// TIA Portal V17 export
// export: Created 2023-04-11T09:33:31.0535455Z, ExportSetting WithDefaults, DisplayName Totally Integrated Automation Portal, DisplayVersion V17 Update 3, DisplayName TIA Portal Openness, DisplayVersion V17 Update 3, DisplayName TIA Portal Version Control Interface, DisplayVersion V17, DisplayName SINAMICS Startdrive Advanced, DisplayVersion V17 Update2, DisplayName SINAMICS Startdrive G130, G150, S120, S150, SINAMICS MV, S210, DisplayVersion V17 Update2, DisplayName SINAMICS Startdrive G110M, G120, G120C, G120D, G120P, G115D, DisplayVersion V17 Update2, DisplayName STEP 7 Professional, DisplayVersion V17 Update 3, DisplayName STEP 7 Safety, DisplayVersion V17, DisplayName WinCC UA Professional, DisplayVersion V17 Update 3
FUNCTION "FC_setStepNameLang" : Bool   // FC18, LAD
{ S7_Optimized_Access := 'TRUE' }
VERSION : 0.1
// stored: AutoNumber true, IsIECCheckEnabled false, SetENOAutomatically false, UDAEnableTagReadback false
   VAR_INPUT
      language : Int;
      text_en : String;
      text_slo : String;
   END_VAR
   VAR_IN_OUT
      index : Int;
      HMI_text : Array[0..2] of String;
   END_VAR
   VAR CONSTANT
      ENG : Int;
      SLO : Int := 1;
   END_VAR
BEGIN

REGION Network 1 (SCL)
   CASE #language OF
       #ENG:  #HMI_text[#index]:=  #text_en;
       #SLO:  #HMI_text[#index] := #text_slo;
   END_CASE;
   #index := #index + 1;

   // zjistit jestli funguje
   //#index := #index AND 3;

   IF #index > 2 THEN
       #index := 2;
   END_IF;
END_REGION
END_FUNCTION
